PROGRAM GarageDoor
VAR
	fbMotion : MoveGarageDoor;
	bActuationButton AT %I* : BOOL; //button that we control through visualization
	bErrorButton AT %I* : BOOL; //button for simulating error
	bDoorOpened : BOOL; //sensor for open door
	bDoorClosed : BOOL; //sensor for close door
	bDoorDriveOverload : BOOL; //sensor for the overload of the door
	bDoorPaused : BOOL; //sensor for pausing the door
	bMotionLight : BOOL; //light that indicates there is motion
	bResetButton : BOOL; //button used to reset the error state
	fPosition : LREAL; //shows the position of the door
	
	bTest1 : BOOL;
	bTest2 : BOOL;
	bTest3 : BOOL;
	
	bTest4 : BOOL;
	bTest5 : BOOL;
	
	bPauseVis : BOOL;
	bErrorVis : BOOL;
	
	bEncOrPwrErr : BOOL; //encoder or power outage error
	bCtrOr24VErr : BOOL; //controller or 24V error
	
	bGearingButton : BOOL;
	
	bAxisMovement : BOOL;
	
	rGearRatio : REAL;
END_VAR

fbMotion.bActuationProgram := bActuationButton;
fbMotion.bError := bErrorButton;
fbMotion.bReset := bResetButton;

bDoorOpened := fbMotion.bOpened;
bDoorClosed := fbMotion.bClosed;
bDoorDriveOverload := fbMotion.bDriveOverload;
bDoorPaused := fbMotion.bPaused;
bMotionLight := fbMotion.bLight;

fPosition := fbMotion.fActPos;

bTest1 := fbMotion.bVis1O;
bTest2 := fbMotion.bVis2O;
bTest3 := fbMotion.bVis3O;

bTest4 := fbMotion.bVis1C;
bTest5 := fbMotion.bVis2C;

bPauseVis := fbMotion.bPauseImg;
bErrorVis := fbMotion.bErrorImg;

bEncOrPwrErr := fbMotion.bEncoderOrPowerErr;
bCtrOr24VErr := fbMotion.bController24VErr;

fbMotion.bGearButton := bGearingButton;

bAxisMovement := fbMotion.bAxisBusy;

fbMotion.rRatioInput := rGearRatio;

fbMotion();

END_PROGRAM

(* stored: Version 1.1.0.1, ProductVersion 3.1.4024.12
   POU GarageDoor: Id {61d642d1-b05b-46ad-9be9-dc37a7c45005}, SpecialFunc None *)
